(* CoDeSys 2.3 export: OBLICZ_KOLIZJE.EXP *)

(* POU OBLICZ_KOLIZJE, ST *)
PROGRAM OBLICZ_KOLIZJE
VAR
END_VAR
Wolne_Prawo := FALSE;
Wolne_Lewo := FALSE;
Wolne_Gora := FALSE;
Wolne_Dol := FALSE;

IF hoz < 20 THEN
    IF Mapa[hoz + 1, ver] = FALSE THEN
        Wolne_Prawo := TRUE;
    END_IF
END_IF


IF hoz > 0 THEN
    IF Mapa[hoz - 1, ver] = FALSE THEN
        Wolne_Lewo := TRUE;
    END_IF
END_IF

IF ver < 15 THEN
    IF Mapa[hoz, ver + 1] = FALSE THEN
        Wolne_Dol := TRUE;
    END_IF
END_IF

IF ver > 0 THEN
    IF Mapa[hoz, ver - 1] = FALSE THEN
        Wolne_Gora := TRUE;
    END_IF
END_IF
END_PROGRAM
